FUNCTION ConvertPressure_Penning : REAL
VAR_INPUT
	penningInt: INT;
END_VAR
VAR
	voltage: LREAL;
END_VAR

//IF voltage < 1.5 OR NOT enabled THEN
//	ConvertPressure_Penning := -1; //ERROR (SENSOR DISCONNECTED??)
//ELSE
//	IF voltage > 9.6 THEN
//		voltage := 9.6;
//	END_IF
//	ConvertPressure_Penning := EXPT(10, ( voltage - 12.86 ) / 1.33 ); // voltage to mbars (formula from Leybold penningvac manual)
//END_IF

//Pfeiffer Penning routine
voltage :=  penningInt / 3276.8;

IF voltage < 2.0 THEN
	ConvertPressure_Penning := 1000; //ERROR (SENSOR DISCONNECTED??)
ELSE
	IF voltage > 8.6 THEN
		voltage := 8.6;
	END_IF
	ConvertPressure_Penning := EXPT(10, ( 1.25 * voltage - 12.75 )); // voltage to mbars (formula from Pfeiffer penningvac IKR 270 manual)
END_IF

END_FUNCTION

(* stored: Version 1.1.0.1, ProductVersion 3.1.4022.16
   POU ConvertPressure_Penning: Id {bd74ec83-25a0-4e21-8bfb-573394af58f7}, SpecialFunc None *)
